FUNCTION_BLOCK FB_NivelSensor IMPLEMENTS I_Analog
VAR_INPUT
END_VAR
VAR_OUTPUT
END_VAR
VAR
	_MaxValue 		: INT;
	_ScaledAnalog 	: INT;
	_AnalogSignal 	: INT;
END_VAR

{warning 'Agregar implementación de propiedad'}
PROPERTY AnalogSignal : INT
GET
AnalogSignal := _AnalogSignal;
END_GET
SET
_AnalogSignal := AnalogSignal;
END_SET
END_PROPERTY

PROPERTY MaxValue : INT
GET
MaxValue := _MaxValue;
END_GET
SET
_MaxValue := MaxValue;
END_SET
END_PROPERTY

{warning 'Agregar implementación de método'}
METHOD Scale : BOOL
ScaledAnalog := AnalogSignal * MaxValue / 1000;
END_METHOD

{warning 'Agregar implementación de propiedad'}
PROPERTY ScaledAnalog : INT
GET
ScaledAnalog := _ScaledAnalog;
END_GET
SET
_ScaledAnalog := ScaledAnalog;
END_SET
END_PROPERTY

END_FUNCTION_BLOCK

(* stored: Version 1.1.0.1, ProductVersion 3.1.4024.12
   POU FB_NivelSensor: Id {0c319140-eb32-41e5-927e-020d0f519e22}, SpecialFunc None
   Property AnalogSignal: Id {f6ad1759-5a15-4ad5-a27c-6dceb5f98753}
   Get Get: Id {78fff54e-39ce-41f6-8d48-de708c5383fa}
   Set Set: Id {8270a37f-bfc0-4af1-90be-f37151cfe08d}
   Property MaxValue: Id {97bbebf4-703c-4100-8637-83ddace2198a}
   Get Get: Id {2ffe5770-0e9e-4a7d-88ab-425a1b837bdc}
   Set Set: Id {d7a18e7a-bfb3-49d3-ac24-3b7fddbf1acc}
   Method Scale: Id {dc2cd368-a319-4da1-8ec9-3648759750a6}
   Property ScaledAnalog: Id {c9d1e697-9b99-4c97-a659-849166b6dc88}
   Get Get: Id {d6c8fa40-6178-4e63-b5b1-248e25f434d8}
   Set Set: Id {51ab4c22-f3ac-418e-8e2a-898e06dcae62} *)
